FUNCTION_BLOCK FB_AR_RANDOM (* Wrapper around FB_RANDOM with AR adapter output plug *)
  (* Standard: 61499-1; Description: Copyright (c) 2026 HR Agrartechnik GmbH This program and the accompanying materials are made available under the terms of the Eclipse Public License 2.0 which is available at https://www.eclipse.org/legal/epl-2.0/ SPDX-License-Identifier: EPL-2.0 *)
  (* Version 1.0, 2026-09-10, Franz Höpfinger, HR Agrartechnik GmbH, Initial Version *)
  PACKAGE adapter::utils;
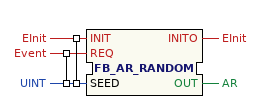
  EVENT_INPUT
    INIT : EInit WITH SEED; (* Initialization Request *)
    REQ WITH SEED; (* Normal Execution Request *)
  END_EVENT
  EVENT_OUTPUT
    INITO : EInit; (* Initialization Confirm *)
  END_EVENT
  VAR_INPUT
    SEED : UINT := 0; (* Seed Value *)
  END_VAR
  PLUGS
    OUT : adapter::types::unidirectional::AR; (* AR adapter output plug *)
  END_PLUGS
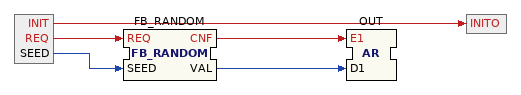
  FBS
    FB_RANDOM : eclipse4diac::utils::FB_RANDOM;
  END_FBS
  EVENT_CONNECTIONS
    INIT TO INITO;
    REQ TO FB_RANDOM.REQ;
    FB_RANDOM.CNF TO OUT.E1;
  END_CONNECTIONS
  DATA_CONNECTIONS
    SEED TO FB_RANDOM.SEED;
    FB_RANDOM.VAL TO OUT.D1;
  END_CONNECTIONS
END_FUNCTION_BLOCK
